Universal Robots PolyScope program: polishing.urp

Program polishing (installation=default directory=/home/ur/ursim-current/programs createdIn=5.14.0 lastSavedIn=5.14.0 robotSerialNumber=20195299999)
Calibrated DH parameters: a=[0, -0.6127, -0.57155, 0, 0, 0]; d=[0.1807, 0, 0, 0.17415, 0.11985, 0.11655]; alpha=[1.570796, 0, 0, 1.570796, -1.570796, 0]; deltaTheta=[0, 0, 0, 0, 0, 0]
InitVariablesNode
Robot Program (runOnlyOnce=false)
  Script file /home/ur/ursim-current/programs/polishing.script
    | # variables
    | global step = 100
    | global radius = 30
    | 
    | # positions (can be defined also as installation variables to store their value)
    | global pa = p[0, 0, 0, 0, 0, 0]
    | global pb = p[0, 0, 0, 0, 0, 0]
    | global pc = p[0, 0, 0, 0, 0, 0]
    | global pd = p[0, 0, 0, 0, 0, 0]
    | 
    | # functions
    | def polish():
    |     d_ab = point_dist(pa, pb)
    | 
    |     repetitions = floor(d_ab / (step/1000))
    |     percentage_ab = (step/1000) / d_ab
    |     percentage_cd = 1 / repetitions
    | 
    |     i = 0
    |     while i < repetitions:
    |         p1 = interpolate_pose(pa, pb, i * percentage_ab)
    |         movel(p1, a=0.1, v=0.2, r=radius/1000)
    | 
    |         p2 = interpolate_pose(pc, pd, i * percentage_cd)
    |         movel(p2, a=0.1, v=0.2, r=radius/1000)
    | 
    |         p3 = interpolate_pose(pc, pd, (i + 1) * percentage_cd)
    |         movel(p3, a=0.1, v=0.2, r=radius/1000)
    | 
    |         p4 = interpolate_pose(pa, pb, (i + 1) * percentage_ab)
    |         movel(p4, a=0.1, v=0.2, r=radius/1000)
    | 
    |         i = i + 2
    | 
    |     end
    | end
  URCap HMI (Robpod HMI URcap, Robpod Cloud) dataModel(robpod.hmi.stop.main.loop=true, robpod.hmi.selected=/home/ur/ursim-current/programs/polishing.hmi)
